(* IEC 61131-3 sources: AXOpen/src/components.keyence.vision/ctrl/src/Axo_SR_750 (part 2) *)

        ///<summary>
		/// Clears the result data.
        ///</summary>
        METHOD PUBLIC ClearResultData : IAxoTaskState
            ClearResultData :=ClearResultDataTask.Invoke(THIS);;
        END_METHOD

        ///<summary>
		/// Triggers the reading sequence and waits for results.
        ///</summary>
        METHOD PUBLIC Read : IAxoTaskState
            VAR_INPUT
                inBank : UINT;
            END_VAR
            VAR_OUTPUT
                result : ARRAY [0..245] OF BYTE;
            END_VAR
            _Bank := inBank;
            result := ResultData.Data;
            Read := ReadTask.Invoke(THIS);
        END_METHOD

        ///<summary>
		/// Triggers the reading sequence and waits for results.
        ///</summary>
        METHOD PUBLIC Tune : IAxoTaskState
            VAR_INPUT
                inBank : UINT;
            END_VAR
            _Bank := inBank;
            Tune := TuneTask.Invoke(THIS);
        END_METHOD

        ///<summary>
		/// Triggers the reading sequence and waits for results.
        ///</summary>
        METHOD PUBLIC Read : IAxoTaskState
            VAR_OUTPUT
                result : ARRAY [0..245] OF BYTE;
            END_VAR
            _Bank := UINT#0;
            result := ResultData.Data;
            Read := ReadTask.Invoke(THIS);
        END_METHOD

        METHOD PRIVATE CallTimers
            VAR_INPUT
                signal : BOOL;
            END_VAR

            _infoTimer.OnDelay(THIS, signal AND Config.InfoTime > LT#0S ,Config.InfoTime);
            _errorTimer.OnDelay(THIS, signal AND Config.ErrorTime > LT#0S , Config.ErrorTime);
        END_METHOD

        METHOD PRIVATE ContinuousReading //TODO
            VAR
                _index : INT;
            END_VAR
            // IF ResultsStatus.ResultsAvailable AND NOT ResultsControl.ResultsAcknowledge AND Results.Code > UINT#0 AND Results.Length > UINT#0 THEN
            //     Messenger.ActivateOnCondition(ULINT#820, Results.Length > TO_UINT(Config.ResultDataSize), eAxoMessageCategory#Error);
            //     TaskMessenger.ActivateOnCondition(ULINT#713, Results.Length > TO_UINT(Config.ResultDataSize), eAxoMessageCategory#Error);
            //     IF Results.Length > TO_UINT(Config.ResultDataSize) THEN
            //         Status.Action.Id := UINT#820;
            //         Status.Error.Id := UINT#713;
            //     ELSE
            //         FOR _index := 0 TO (TO_INT(Results.Length) - INT#1) DO
            //             ResultData.Data[_index] := _data_in[_index + 8];
            //         END_FOR;
            //         FOR _index := TO_INT(Results.Length) TO 245 DO
            //             ResultData.Data[_index] := BYTE#0;
            //         END_FOR;
            //         ResultData.DataChanged := NOT ResultData.DataChanged ;
            //         Status.Action.Id := UINT#120;
            //     END_IF;
            // END_IF;

            // ResultsControl.ResultsAcknowledge := ResultsStatus.ResultsAvailable;
            ;
        END_METHOD

        ///<summary>
		/// Custom logic for the manual control.
        ///</summary>
        METHOD PROTECTED OVERRIDE ManualControl
            ;
        END_METHOD

        ///<summary>
		/// Restores this instance to its initial state.
        ///</summary>
        METHOD PUBLIC OVERRIDE Restore
            VAR
                _index : INT;
            END_VAR
            Status.Action.Id := UINT#0;
            Status.Error.Id  := UINT#0;
            Messenger.Restore();
            TaskMessenger.Restore();

            ClearResultDataTask.Restore();
            ReadTask.Restore();
            TuneTask.Restore();

            LatchAndErrorClearControl.ResultDataLatch               :=  FALSE;
            LatchAndErrorClearControl.ErrorClear                    :=  FALSE;
            OperationInstructionControl.ReadRequest                 :=  FALSE;
            OperationInstructionControl.PresetRequest               :=  FALSE;
            OperationInstructionControl.RegisterPresetDataRequest	:=  FALSE;
            OperationInstructionControl.TuneRequest	                :=  FALSE;
            CompletionClearControl.ReadCompleteClear	            :=  FALSE;
            CompletionClearControl.PresetCompleteClear	            :=  FALSE;
            CompletionClearControl.RegisterPresetDataCompleteClear	:=  FALSE;
            CompletionClearControl.TuneCompleteClear	            :=  FALSE;
            CompletionClearControl.EXT_RequestCompleteClear	        :=  FALSE;
            ParameterBankNumber.BankNumberRegister	                :=  UINT#0;
            User.UserDataSize                                       :=  UINT#0;

            _prevResultDataReadyCount                               :=  UINT#0;
            _prevResultDataUpdateCount                              :=  UINT#0;
            _resultString                                           :=  '';
            ReadData.ResultDataSize                                 :=  UINT#0;

            FOR _index := 0 TO 245 DO
                ResultData.Data[_index] := BYTE#0;
            END_FOR;

            IF NOT HandshakeAndGeneralErrorStatus.GeneralError THEN
                Status.Action.Id := UINT#50;
                RestoreTask.DoneWhen(TRUE);
            END_IF;
        END_METHOD
    END_CLASS
END_NAMESPACE
